{attribute 'qualified_only'}
{attribute 'strict'}
{attribute 'to_string'}
TYPE EPowerIlluminationFlow :
(
	HS := 1,
	HT
);
END_TYPE

(* stored: Version 1.1.0.1, ProductVersion 3.1.4024.4
   DUT EPowerIlluminationFlow: Id {c4387d13-332f-4e8c-9c0d-0cbef6adfaaa} *)
